{attribute 'call_after_init'}
FUNCTION_BLOCK FB_ChillerLoop_Test EXTENDS FB_TestSuite
VAR_INPUT
END_VAR
VAR_OUTPUT
END_VAR
VAR
END_VAR

TemperatureErrorTriggers();
TemperatureErrorReturnsToNormal();
NoError();
//OperatorOverrideResets();

METHOD NoError
VAR
	fbChillerLoop : FB_ChillerLoop;
END_VAR
TEST('NoChillerLoopError');

fbChillerLoop(bLoopTempSW := TRUE);
AssertFalse(fbChillerLoop.bError, 'Error fasely detected');

TEST_FINISHED();
END_METHOD

METHOD OperatorOverrideResets
VAR
	fbChillerLoop : FB_ChillerLoop;
END_VAR
(*
TEST('OperatorOverrideResets');

fbChillerLoop(bLoopTempSW := FALSE);
fbChillerLoop.bOperatorOverride := TRUE;
AssertTrue(fbChillerLoop.bOperatorOverride, 'Operator override failed to set');

// Operator override should reset uner normal temperature conditions.
fbChillerLoop(bLoopTempSW := TRUE);
AssertFalse(fbChillerLoop.bOperatorOverride, 'Operator override failed to reset');

TEST_FINISHED();
*)
END_METHOD

METHOD TemperatureErrorReturnsToNormal
VAR
	fbChillerLoop : FB_ChillerLoop := F_ChillerLoop_Error();
END_VAR
TEST('TemperatureErrorReturnsToNormal');

// Chiller loop should return to normal state when inputs go back to normal
fbChillerLoop(bLoopTempSW := TRUE);
AssertFalse(fbChillerLoop.bError, 'Temperature error did not go back to normal');

TEST_FINISHED();
END_METHOD

METHOD TemperatureErrorTriggers
VAR
	fbChillerLoop : FB_ChillerLoop := F_ChillerLoop_Error();
END_VAR
TEST('TemperatureErrorTriggers');

AssertTrue(fbChillerLoop.bError, 'Temperature error did not trigger');

TEST_FINISHED();
END_METHOD

END_FUNCTION_BLOCK

(* stored: Version 1.1.0.1, ProductVersion 3.1.4022.17
   POU FB_ChillerLoop_Test: Id {8ac89975-cd8d-49dd-8cf3-ec426456b1c0}, SpecialFunc None
   Method NoError: Id {dd242c58-8b42-478d-9d9b-26e741e96a35}
   Method OperatorOverrideResets: Id {dc3a5974-2d91-46f0-b32a-8ef644cca320}
   Method TemperatureErrorReturnsToNormal: Id {fdc4b03e-9d62-4e4f-aedd-88c595d75147}
   Method TemperatureErrorTriggers: Id {f317dc99-d319-4c6c-92d4-c5a67e245736} *)
